FUNCTION_BLOCK PusherResetDelay (* Basic Function Block Type *)
  (* Standard: 61499-2 *)
  (* Version 0.0, 21.06.2022, david, WBK hackaton, Template *)
  PACKAGE Main;
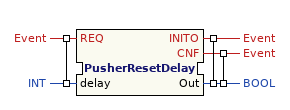
  EVENT_INPUT
    REQ WITH delay; (* Normal Execution Request *)
  END_EVENT
  EVENT_OUTPUT
    INITO WITH Out; (* Initialization Confirm *)
    CNF WITH Out; (* Execution Confirmation *)
  END_EVENT
  VAR_INPUT
    delay : INT; (* Numer ob ticks to delay event activation *)
  END_VAR
  VAR_OUTPUT
    Out : BOOL; (* Output event qualifier *)
  END_VAR
  VAR
    tickCounter : INT := 0;
  END_VAR
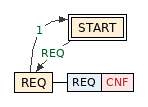
  EC_STATES
    START; (* Initial State *)
    REQ : REQ -> CNF; (* Normal execution *)
  END_STATES
  EC_TRANSITIONS
    START TO REQ := REQ;
    REQ TO START := 1;
  END_TRANSITIONS
  ALGORITHM INIT IN ST: (* Initialization algorithm *)
;
  END_ALGORITHM
  ALGORITHM REQ IN ST: (* Normally executed algorithm *)
IF tickCounter<delay THEN
	tickCounter:=tickCounter+1;
	Out:=0;
ELSE
	tickCounter:=0;
	Out:=1;
END_IF
;
  END_ALGORITHM
END_FUNCTION_BLOCK
